// TIA Portal V20 export
VAR_GLOBAL   // PLC tag table "LConSMC_Warnings"
END_VAR
VAR_GLOBAL CONSTANT   // user constants
   LCON_WARNING_WINDER_MAX_VELOCITY_EXCEEDED : DWord := 16#5105_4004;   // Warning that the output is limited. The input line velocity is limited to config.maxVelocity
   LCON_WARNING_SECTIONAL_DRIVE_OUTPUT_LIMITED : DWord := 16#7102_4000;   // Warning that the output is limited. The torque limits are limited between 0-200%
   LCON_WARNING_SECTIONAL_DRIVE_TORQUE_PRECONTROL_DISABLED : DWord := 16#7102_4005;   // The torque precontrol has been disabled internally if the sign of the torque limit changes for torque controlled modes
   LCON_WARNING_WINDER_TORQUE_PRECONTROL_ACTIVE : DWord := 16#5105_4002;   // No telegram 750 is connected but torque precontrol is selected at the FB (adjustment <> 0.0). Torque precontrol is deactivated internally.
   LCON_WARNING_WINDER_RUN_AWAY_DETECTED : DWord := 16#5105_4006;   // In a torque controlled tension mode the deviation between line velocity setpoint and actual circumference velocity has exceeded a limit. The friction and/or acceleration torque pre-control values might be invalid and have been disabled.
   LCON_WARNING_SECTIONAL_DRIVE_RUN_AWAY_DETECTED : DWord := 16#7102_4006;   // In a torque controlled tension mode the deviation between line velocity setpoint and actual circumference velocity has exceeded a limit. The friction and/or acceleration torque pre-control values might be invalid and have been disabled.
   LCON_WARNING_WINDER_TORQUE_PRECONTROL_DISABLED : DWord := 16#5105_4005;   // The torque precontrol has been disabled internally if the sign of the torque limit changes for torque controlled modes
   LCON_WARNING_WINDER_NO_WEB_BREAK_DETECTION_POSSIBLE : DWord := 16#5105_4003;   // Web break detection not possible in this control mode
   LCON_WARNING_WINDER_OUTPUT_LIMITED : DWord := 16#5105_4000;   // Warning that the output is limited. The torque limits are limited between 0-200%
   LCON_WARNING_CALC_TARGET_DIAM_STOP_COND_OUTPUT_LIMITED : DWord := 16#4004_4000;   // Warning that the output is limited
   LCON_WARNING_FRICTION_V2_OUTPUT_LIMITED : DWord := 16#3113_4000;   // Warning that the output is limited
   LCON_WARNING_SECTIONAL_DRIVE_MAX_VELOCITY_EXCEEDED : DWord := 16#7102_4004;   // Warning that the output is limited. The input line velocity is limited to config.maxVelocity
   LCON_WARNING_TABLE_CHAR_NO_VALUE_FOUND : DWord := 16#0106_4001;   // Warning that no value is found
END_VAR
